FUNCTION_BLOCK Q_ActiveMask (* Command change active mask( Part 6 - F.34 ) *)
  (* Standard: ISO 11783-6; Description: This command is used to change the active mask of a working set to either a data or an alarm mask object. Return values iso_s16 - E_NO_ERR - OK - E_OVERFLOW - buffer overflow - E_NOACT - Command not possible in current state - E_NO_INSTANCE - No VT client available *)
  (* Version 1.0, 2022-07-08, franz *)
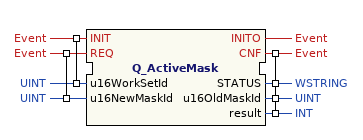
  EVENT_INPUT
    INIT WITH u16WorkSetId; (* Service Initialization *)
    REQ WITH u16NewMaskId; (* Service Request *)
  END_EVENT
  EVENT_OUTPUT
    INITO; (* Initialization Confirm *)
    CNF WITH STATUS, u16OldMaskId, result, u16OldMaskId; (* Confirmation of Requested Service *)
  END_EVENT
  VAR_INPUT
    u16WorkSetId : UINT; (* WorkingSet Object ID *)
    u16NewMaskId : UINT; (* Object ID of new active (data/alarm)-mask *)
  END_VAR
  VAR_OUTPUT
    STATUS : WSTRING; (* Service Status *)
    u16OldMaskId : UINT; (* Object ID of old active (data/alarm)-mask *)
    result : INT; (* retval see description *)
  END_VAR
END_FUNCTION_BLOCK
